Staubli VAL3: onStart.pgx

public program onStart(string& x_sItem[])
begin
  //
  // Done on the start of the kernel
  //
end
